Staubli VAL3: startAreaTest.pgx

public program startAreaTest()
begin
  // start area test state machine
  nAreaTestState=10
end
